(*

.. <legal notes>

legal notes
=================
| SPDX-FileCopyrightText: © 2025 Oleksandr Tiutyk <trofimich@gmail.com>
| SPDX-License-Identifier: LGPL-3.0-only
| For details check: LGPL-3.0-only_

.. _LGPL-3.0-only: https://www.gnu.org/licenses/lgpl-3.0.en.html

.. </legal notes>

*)

INTERFACE IProcess EXTENDS IObject

{attribute 'monitoring' := 'call'}
{attribute 'OPC.UA.DA.Property' := '1'}
{attribute 'OPC.UA.DA.Access' := '1'}
PROPERTY Error : BOOL
GET
END_GET
END_PROPERTY

{attribute 'monitoring' := 'call'}
{attribute 'OPC.UA.DA.Property' := '1'}
{attribute 'OPC.UA.DA.Access' := '1'}
PROPERTY ErrorMessage : REFERENCE TO ERROR_MESSAGE
GET
END_GET
END_PROPERTY

METHOD Execute
END_METHOD

{attribute 'monitoring' := 'call'}
{attribute 'OPC.UA.DA.Property' := '1'}
{attribute 'OPC.UA.DA.Access' := '1'}
PROPERTY Name : WSTRING
GET
END_GET
END_PROPERTY

{attribute 'monitoring' := 'call'}
{attribute 'OPC.UA.DA.Property' := '1'}
{attribute 'OPC.UA.DA.Access' := '1'}
PROPERTY Running : BOOL
GET
END_GET
END_PROPERTY

METHOD Start
END_METHOD

{attribute 'monitoring' := 'call'}
{attribute 'OPC.UA.DA.Property' := '1'}
{attribute 'OPC.UA.DA.Access' := '1'}
PROPERTY StateChanged : BOOL
GET
END_GET
END_PROPERTY

END_INTERFACE

(* stored: Version 1.1.0.1
   Itf IProcess: Id {44e3ce8b-ac1f-4d7c-a60d-08ecae2ae96e}
   Property Error: Id {ec720c04-807f-445f-ab2a-39f8da91a7e2}
   Get Get: Id {34fec23a-5830-4fef-a20d-8e34142e370a}
   Property ErrorMessage: Id {271524ea-f71b-44d8-9e2a-c8365de6d7eb}
   Get Get: Id {679dc1f0-6f58-485c-8248-dbc0713e8e6d}
   Method Execute: Id {ce1f820d-f7df-4937-80f2-bfbc5db53fec}
   Property Name: Id {ef024ee8-bb4e-475f-a01f-56d9aa5ebcfb}
   Get Get: Id {400a1239-4405-4d0c-a905-63436eccf146}
   Property Running: Id {51e451a4-81f2-47fb-a17a-20d4804995fb}
   Get Get: Id {8af8039c-c89d-41e0-9d7d-145433c29bed}
   Method Start: Id {631e33ee-b37e-460c-8e59-222465f56e8a}
   Property StateChanged: Id {b4cbb541-af3a-4b44-bf2d-1848d01f548c}
   Get Get: Id {4150f858-b1df-4796-959f-aa93a001e34e} *)
